(********************* G.D S.p.A. - Technical Department ***********************************
This program has been generated automatically from Application Designer DE&F
********************************************************************************************)
PROGRAM dbg_csp_case_closing_ls_upper
VAR
  axis_shd : axis_shadow;
END_VAR

_objects_manager();

IF	g_application_status <> APPLICATION_STATUS_RUNNING
THEN
	RETURN;
END_IF

CASE process_get_mode(CONVERSION_this := dbg_root.prc) OF
	MODE_ABSENT,
	MODE_INACTIVE:
		RETURN;
	MODE_TEST:
		RETURN;
END_CASE

ACTION _objects_manager:
IF	objects_initialization()
THEN
	axis_shadow_init(
		sim_mode:= SHADOW_SIMULATION_MODE_AUTOMATIC, 
		father:= csp_case_closing_ls_upper.axis, 
		process:= dbg_root.prc, 
		CONVERSION_this:= axis_shd);

	RETURN;
END_IF

IF	objects_running()
THEN
	axis_shadow_cycle(axis_shd);
END_IF
END_ACTION

END_PROGRAM

(* stored: Version 1.1.0.1, ProductVersion 3.1.4022.12
   POU dbg_csp_case_closing_ls_upper: Id {60b79352-762a-4b6f-a654-2d0f33f5195b}, SpecialFunc None
   Action _objects_manager: Id {73a1d9ad-d0b1-4b8a-9fb4-415469e7f1c5} *)
